(*
SPDX-FileCopyrightText: © 2026 Oleksandr Tiutyk <trofimich@gmail.com>
SPDX-License-Identifier: MIT
License: https://opensource.org/license/mit
*)

(*!
<summary>Reports a required argument that the caller considers unspecified.</summary>
<description>
The caller detects the invalid argument. Throw records a diagnostic message and source metadata; it does not
inspect the actual argument or decide which types are supported. Dynamic instances belong to the current task
memory manager until cleanup.
</description>
*)
INTERFACE IArgumentNotSpecifiedException EXTENDS IGeneralException

(*!
<summary>Builds the argument diagnostic and propagates this exception.</summary>
<description>
Call in the owning cyclic task, not during FB_init. Captures message, source and timestamps with zero error
code and no inner cause. Supplied names are copied into the message; no caller storage is retained. Allocation
failure follows the shared terminal memory mechanism.
</description>
<param name="argumentName">Name of the argument rejected by the caller.</param>
*)
METHOD Throw
VAR_INPUT
	sourceNamespaceName : STRING;
	sourceClassName : STRING;
	sourcePOUName : STRING;
	sourcePosition : STRING;
	argumentName : STRING;
END_VAR
END_METHOD

END_INTERFACE

(* stored: Version 1.1.0.1
   Itf IArgumentNotSpecifiedException: Id {8d1dcd2c-ca51-4f93-8b0f-4c12ec4ce6a4}
   Method Throw: Id {170f19d7-15b2-43f5-807c-aef9f4d86d53} *)
